VAR_GLOBAL
	gTimeZoneOffset	: DINT;			// Time Zone Offset from UTC
	gCurrentTime	: TimeStamp;	// Current Time for Station
END_VAR

(* stored: Version 1.1.0.1, ProductVersion 3.1.4024.9
   GVL Global_Variables: Id {5725dc71-9437-4faa-b9ac-8413153f35a5} *)
